// TwinCAT 3 PLC project nadaCAT
// ProgramVersion: 3.1.4024.0
// libraries:
//   Tc2_MC2, * (Beckhoff Automation GmbH)
//   Tc2_MC2_Drive, * (Beckhoff Automation GmbH)
//   Tc2_Standard, * (Beckhoff Automation GmbH)
//   Tc2_System, * (Beckhoff Automation GmbH)
//   Tc2_TcpIp, * (Beckhoff Automation GmbH)
//   Tc2_Utilities, * (Beckhoff Automation GmbH)
//   Tc3_Module, * (Beckhoff Automation GmbH)
//   VisuDialogs, * (System)
//   VisuSymbols,3.5.10.0,System
// project tree:
//   DUTs/Enums/ E_CommandList.TcTLEO, E_ServoState.TcTLEO (not stored), E_TCPState.TcTLEO
//   DUTs/Hardware/ EL1008.TcDUT (not stored), EL2008.TcDUT (not stored)
//   DUTs/Structs/ dutCommand.TcDUT (not stored), dutResponse.TcDUT, mcInterface.TcDUT, mcOutputs.TcDUT, stConfigParams.TcDUT, stIOinput.TcDUT, stIOoutput.TcDUT, stServoInterface.TcDUT, stStateTransitions.TcDUT (not stored)
//   / GlobalTextList.TcGTLO, PlcTask.TcTTO, Visualization Manager.TcVMO (not stored), VISU_TASK.TcTTO (not stored)
//   GVLs/ gvlMotion.TcGVL, gvlIO.TcGVL, gvlSystem.TcGVL, gvlServo.TcGVL (not stored)
//   POUs/FBs/ FB_AutoMotionControl.TcPOU, FB_ManualMotionControl.TcPOU, FB_ManualMotionControlNew.TcPOU, FB_ManualStateMachine.TcPOU (not stored), FB_TCPServer.TcPOU (not stored), sfc_TCPServer.TcPOU (not stored)
//   POUs/ MAIN.TcPOU
//   POUs/PRGs/ prgMotion.TcPOU (not stored), prgIO.TcPOU, prgSystem.TcPOU, prgTCPComm.TcPOU (not stored)
//   VISUs/ Main.TcVIS (not stored)
//   VISUs/Templates/ MotorFaceplate.TcVIS, MotorFaceplate2.TcVIS (not stored), SysPanel.TcVIS (not stored)
// real-time tasks:
//   TASK PlcTask: cycle T#10ms, priority 20, ADS port 350
//   TASK VISU_TASK: cycle T#200000us, priority 30, ADS port 351
// motion (NC):
//   TASK NC-Task 1 SAF: cycle T#2ms, priority 4, ADS port 501
//   TASK NC-Task 1 SVB: cycle T#10ms, priority 8, ADS port 511
//   AXIS Bank1 (id 4)
//     Dynamic: AccelerationMaximum=1000, DecelerationMaximum=1000, Acceleration=250, Deceleration=250, Jerk=1000, FastAcceleration=10000, FastDeceleration=10000, FastJerk=10000
//     Velo: Maximum=450
//     OtherSettings: AllowMotionCmdToSlave=true
//     encoder EncType=19
//       EncPara: ScaleFactorNumerator=10, ScaleFactorDenominator=3600000, Offset=2.25188333333333, Inverse=true, MaxCount=#xffffffff, ReferenceSystem=3
//         SoftEndMinControl: Enable=true
//         SoftEndMaxControl: Enable=true, Range=860
//     drive DrvType=16
//       DrvPara: Inverse=true, MaxCount=#xffffffff, DriveControlDWord=#x00020000
//         Analog: TorqueSetpointScale=10, ScaleFactorActTorque=0.1
//         TimeComp: TaskDelayCycles=1
//     controller CtrType=1
//       CtrPara: PriorControlFactor=1
//         Observer: BandWidth=20
//   AXIS Virtual (id 2)
//     OtherSettings: AllowMotionCmdToSlave=true
//     encoder EncType=1
//       SoftEndMinControl: Enable=true, Range=-0.1
//       SoftEndMaxControl: Enable=true, Range=860
//     drive DrvType=5
//       Analog: TorqueSetpointScale=10, ScaleFactorActTorque=0.1
//       TimeComp: TaskDelayCycles=1
//     controller CtrType=1
//       CtrPara: PriorControlFactor=1
//         Observer: BandWidth=20
// I/O:
//   DEVICE Device 1 (EtherCAT) (disabled), AmsNetId 192.168.5.101.2.1
//     Drive 1 (IndraDrive MPB20/21 CoE) [IndraDrive MPB20/21 CoE]
//       modules: Module 1 (Cyclic sync position mode)
// variable links:
//   NC-Task 1 SAF/Axes/Bank1 <-> Device 1 (EtherCAT)/Drive 1 (IndraDrive MPB20/21 CoE)
//     Drive/Inputs/In/nDcOutputTime <-> InfoData/DcOutputShift
//     Drive/Inputs/In/nState1 <-> Module 1 (Cyclic sync position mode)/Transmit PDO Mapping Parameter/CiA402: Statusword
//     Drive/Inputs/In/nState2 <-> Module 1 (Cyclic sync position mode)/Transmit PDO Mapping Parameter/CiA402: Statusword @bit 8
//     Drive/Inputs/In/nState4 @bit 1 <-> WcState/InputToggle
//     Drive/Inputs/In/nState4 <-> WcState/WcState
//     Drive/Outputs/Out/nCtrl1 <-> Module 1 (Cyclic sync position mode)/Receive PDO Mapping Parameter/CiA402: Controlword
//     Drive/Outputs/Out/nCtrl2 <-> Module 1 (Cyclic sync position mode)/Receive PDO Mapping Parameter/CiA402: Controlword @bit 8
//     Drive/Outputs/Out/nDataOut1 <-> Module 1 (Cyclic sync position mode)/Receive PDO Mapping Parameter/CiA402: Target position
//     Enc/Inputs/In/nDataIn1 <-> Module 1 (Cyclic sync position mode)/Transmit PDO Mapping Parameter/CiA402: Position actual value
//     Enc/Inputs/In/nDcInputTime <-> InfoData/DcInputShift
//     Enc/Inputs/In/nState4 @bit 1 <-> WcState/InputToggle
//     Enc/Inputs/In/nState4 <-> WcState/WcState
//   nadaCAT/nadaCAT Instance <-> NC-Task 1 SAF/Axes/Virtual
//     PlcTask Inputs/ServoGVLs.servo1Interface.ioAxisRef.NcToPlc <-> Outputs/ToPlc
//     PlcTask Outputs/ServoGVLs.servo1Interface.ioAxisRef.PlcToNc <-> Inputs/FromPlc

CONFIGURATION nadaCAT
    RESOURCE PLC ON TwinCAT3
        TASK PlcTask(INTERVAL := T#10ms, PRIORITY := 20);
        PROGRAM MAIN WITH PlcTask : MAIN;
    END_RESOURCE
END_CONFIGURATION

// ---- DUTs/Enums/E_CommandList.TcTLEO
{attribute 'qualified_only'}
{attribute "to_string'}
TYPE E_CommandList :
(
	ERR := -1,
	NULL := 0,
	LIST,
	HOM,
	SCAN,
	MTP,
	MOVA,
	MOVR,
	STAT,
	CALIB,
	PARAM
);
END_TYPE
//  ERR = '-1'

// ---- DUTs/Enums/E_TCPState.TcTLEO
{attribute 'qualified_only'}
{attribute 'strict'}
TYPE E_TCPState :
(
	enum_member := 0
);
END_TYPE

// ---- DUTs/Structs/dutResponse.TcDUT
TYPE dutResponse :
STRUCT
END_STRUCT
END_TYPE

// ---- DUTs/Structs/mcInterface.TcDUT
TYPE mcInterface :
STRUCT
	bBusy				: BOOL;
	bActive				: BOOL;
	bCommandAborted		: BOOL;
	bError				: BOOL;
	iErrorID			: UDINT;
END_STRUCT
END_TYPE

// ---- DUTs/Structs/mcOutputs.TcDUT
TYPE mcOutputs :
STRUCT
	Status			: BOOL;
	Done			: BOOL;
	Busy			: BOOL;
	Active			: BOOL;
	CommandAborted	: BOOL;
	Error			: BOOL;
	ErrorID			: UDINT;
	
END_STRUCT
END_TYPE

// ---- DUTs/Structs/stConfigParams.TcDUT
TYPE stConfigParams :
STRUCT
	iSpeed		: INT;  		// Stocker speed
	iAccel		: INT;  		// Stocker acceleration
	iDecel		: INT;  		// Stocker deceleration
	sRamp		: STRING(255);  // Stocker ramp style
	iPodPos		: INT;  		// Stocker pod position, given pod
	iScStart	: INT;  		// Stocker start scanning position
	iScEnd		: INT;  		// Stocker end scanning position
	iScThick	: INT;  		// Average wafer thickness
	iScExclLo	: INT;  		// Low wafer exclusion zone (in percent)
	iScExclHi	: INT;			// High wafer exclusion zone (in percent)
	iPdSlot		: INT;  		// Pod slot count
	iPdBtm		: INT;  		// Pod bottom slot position
	iPdTop		: INT;  		// Pod top slot position

END_STRUCT
END_TYPE

// ---- DUTs/Structs/stIOinput.TcDUT
TYPE stIOinput :
STRUCT
// ~~~~~ Input Signals ~~~~~
	// Drive CoE
	coeProbe1Signal			: WORD;
	coeProbe1PosLatch		: WORD;
	coeProbe1NegLatch		: WORD;
	
	// Hardware Signals
	Rack1Slot2				: EL1008;
	
END_STRUCT
END_TYPE

// ---- DUTs/Structs/stIOoutput.TcDUT
TYPE stIOoutput :
STRUCT
// ~~~~~ Output Signals ~~~~~
	// Drive CoE
	coeProbingCycleCommand	: WORD;
	coeProbe1Enable			: WORD;
	
	// Hardware Signals
	Rack1Slot2				: EL1008;
END_STRUCT
END_TYPE

// ---- DUTs/Structs/stServoInterface.TcDUT
TYPE stServoInterface :
STRUCT
	/// In_Outs
	ioAxisRef			: Axis_Ref;
	/// Inputs
	bDriveEnable		: BOOL;
	bStopMotion			: BOOL;
	bFaultReset			: BOOL;
	bTriggerMove		: BOOL;
	bJogFWD				: BOOL;
	bJogRev				: BOOL;
	bHome				: BOOL;
	bDemoModeActive		: BOOL;
	bDemoModeStart		: BOOL;
	bDemoModeStop		: BOOL;
	iMotionSelect		: INT;
	rSpeed				: REAL;
	rAccelDecel			: REAL;
	rPosition			: REAL;
	/// Outputs
	bDriveEnabled		: BOOL;
	bStopped			: BOOL;
	bFaulted			: BOOL;
	bMoving				: BOOL;
	bNotMoving			: BOOL;
	bAtHome				: BOOL;
	bAccelerating		: BOOL;
	bDecelerating		: BOOL;
	bDemoModePermissive	: BOOL;
	bInposition			: BOOL;
	bInVelocity			: BOOL;
	rActualSpeed		: REAL;	
	rActualPosition		: REAL;

	
END_STRUCT
END_TYPE

// ---- GVLs/gvlMotion.TcGVL
{attribute 'qualified_only'}
VAR_GLOBAL
// Manual Control
servo1			: FB_ManualMotionControlNew;
bank1			: FB_AutoMotionControl;
manualMode 		: BOOL := TRUE;
autoMode		: BOOL;

// Server Control
cmdData 		: dutCommand;
bEnableDrive	: BOOL := FALSE;
bStartDrive		: BOOL := FALSE;
bTriggerDefault : BOOL := FALSE;
bInterlockOK	: BOOL := TRUE;
mcBankAxis		: stServoInterface;
driveStatus 	: ST_AxisStatus;	
END_VAR

// ---- GVLs/gvlIO.TcGVL
{attribute 'qualified_only'}
VAR_GLOBAL
	/// Inputs
	stInputs	:	stIOinput;
	/// Outputs
	stOutputs	: 	stIOoutput;
	
	bHomeSwitch: BOOL;
END_VAR

// ---- GVLs/gvlSystem.TcGVL
{attribute 'qualified_only'}
VAR_GLOBAL
	iTaskIdx 	: DINT;
	bFirstCycle : BOOL;
END_VAR

// ---- POUs/MAIN.TcPOU
PROGRAM MAIN
VAR

END_VAR

// System Control
gvlSystem.iTaskIdx  := GETCURTASKINDEXEX();
prgSystem(iTaskIdx 	:= gvlSystem.iTaskIdx,
	   bFirstCycle  := gvlSystem.bFirstCycle);

// IO (comment for simulation)
//prgIO();
	   
// TCP Connection
prgTCPComm(cmdData => gvlMotion.cmdData);

// Motion Control
prgMotion(
	cmdData:= gvlMotion.cmdData, 
	bAutoEnableDrive:= gvlMotion.bEnableDrive, 
	bAutoStartDrive:= gvlMotion.bStartDrive, 
	bAutoInterlockOK:= gvlMotion.bInterlockOK, 
	bAutoTriggerDefault:= gvlMotion.bTriggerDefault, 
	autoDriveStatus=> gvlMotion.driveStatus, 
	cmdResponse=>, 
	arrServoInterface:= gvlServo.arrServoInterface);

END_PROGRAM

// ---- POUs/PRGs/prgSystem.TcPOU
PROGRAM prgSystem
VAR_IN_OUT
	iTaskIdx		: DINT;
	bFirstCycle		: BOOL;
END_VAR

// Scan Control
bFirstCycle := TwinCAT_SystemInfoVarList._TaskInfo[iTaskIdx].FirstCycle;

// Mode Control
gvlMotion.autoMode := NOT gvlMotion.manualMode;

END_PROGRAM

// ---- POUs/FBs/FB_ManualMotionControlNew.TcPOU
FUNCTION_BLOCK FB_ManualMotionControlNew
VAR_INPUT
	iCmdMova		:	INT := 0;
	iCmdMovr		: 	INT := 0;
	bEnableDrive	:   BOOL;
	bStartDrive		: 	BOOL;
	bRunOnce		:   BOOL := TRUE;
END_VAR
VAR_OUTPUT
	driveStatus	: ST_AxisStatus;
END_VAR
VAR_IN_OUT
	mcBankAxis	: stServoInterface;
END_VAR

VAR
	eState					: E_ServoState;
	demoState				: FB_ManualStateMachine;
	servoPower				: MC_Power;
	servoBuffer				: MC_BufferMode := MC_Aborting;
	servoReset				: MC_Reset;
	servoHome				: MC_Home;
	servoStatus				: MC_ReadStatus;
	servoSetPosition		: MC_SetPosition;
	servoJog				: MC_Jog;
	servoStop				: MC_Stop;
	servoMoveAbsolute		: MC_MoveAbsolute;
	servoMoveRelative		: MC_MoveRelative;
	servoMoveVelocity		: MC_MoveVelocity;
	jogErrorID				: UDINT;
	errorStop: BOOL;
	disabled: BOOL;
	stopping: BOOL;
	discreteMotion: BOOL;
	continuousMotion: BOOL;
	syncMotion: BOOL;
	homing: BOOL;
	constVelocity: BOOL;
	accel: BOOL;
	decel: BOOL;
	status: ST_AxisStatus;
	powerInterface 		: mcInterface;
	resetInterface		: mcInterface;
	homeInterface		: mcInterface;
	jogInterface		: mcInterface;
	stopInterface		: mcInterface;
	moveAbsInterface	: mcInterface;
	moveRelInterface	: mcInterface;
	moveVelInterface	: mcInterface;
	statusInterface		: mcInterface;
	
	// State Machine Variables
	startCycle			: BOOL;
	continueToTop		: BOOL;
	continueToBottom	: BOOL;
	endAtTop			: BOOL;
	endAtBottom			: BOOL;
	moveBottomTrig			: BOOL;
	moveTopTrig				: BOOL;
	
	demoModePermissive	: BOOL;
	demoModeRun			: BOOL;
	bottomComplete		: BOOL;
	topComplete			: BOOL;
	
	servoMoveBottom		: MC_MoveAbsolute;
	servoMoveTop		: MC_MoveAbsolute;
	servoEstop			: MC_Halt;
	
	demoModePermissivesdf: INT;
END_VAR

// ~~~~ Manual FB Inits ~~~~
// Status
servoStatus(
	Axis:= mcBankAxis.ioAxisRef, 
	Enable:= TRUE, 
	Valid=> , 
	Busy=> statusInterface.bBusy, 
	Error=> statusInterface.bError, 
	ErrorID=> statusInterface.iErrorID, 
	ErrorStop=> errorStop, 
	Disabled=> disabled, 
	Stopping=> stopping, 
	StandStill=> mcBankAxis.bNotMoving, 
	DiscreteMotion=> discreteMotion, 
	ContinuousMotion=> continuousMotion, 
	SynchronizedMotion=> syncMotion, 
	Homing=> homing, 
	ConstantVelocity=> mcBankAxis.bInVelocity, 
	Accelerating=> mcBankAxis.bAccelerating, 
	Decelerating=> mcBankAxis.bDecelerating, 
	Status=> status);

// Enable
servoPower(
	Axis:= mcBankAxis.ioAxisRef, 
	Enable:= mcBankAxis.bDriveEnable, 
	Enable_Positive:=TRUE , 
	Enable_Negative:=TRUE , 
	Override:=100.0 , 
	BufferMode:=servoBuffer , 
	Options:= servoPower.Options, 
	Busy=> powerInterface.bBusy, 
	Active=> powerInterface.bActive, 
	Error=> powerInterface.bError, 
	ErrorID=> powerInterface.iErrorID);
// Init Stop
servoStop(
	Axis:= mcBankAxis.ioAxisRef, 
	Execute:=mcBankAxis.bStopMotion , 
	Deceleration:= 100, 
	Jerk:=100 , 
	Options:= servoStop.Options, 
	Busy=>stopInterface.bBusy , 
	Active=>stopInterface.bActive , 
	CommandAborted=>stopInterface.bCommandAborted , 
	Error=> stopInterface.bError, 
	ErrorID=> stopInterface.iErrorID);

// Init HOM
servoHome(
	Axis:= mcBankAxis.ioAxisRef, 
	Execute:= mcBankAxis.bHome, 
	Position:=0.0 , 
	HomingMode:= MC_DefaultHoming, 
	BufferMode:= servoBuffer, 
	bCalibrationCam:=gvlIO.bHomeSwitch , 
	Busy=>homeInterface.bBusy , 
	Active=> homeInterface.bActive, 
	CommandAborted=>homeInterface.bCommandAborted , 
	Error=>homeInterface.bError , 
	ErrorID=> homeInterface.iErrorID);

// Init JOG
servoJog(
	Axis:= mcBankAxis.ioAxisRef, 
	JogForward:= mcBankAxis.bJogFWD, 
	JogBackwards:= mcBankAxis.bJogRev, 
	Mode:= servoJog.Mode, 
	Position:=5 , 
	Velocity:= 1, 
	Acceleration:= 250, 
	Deceleration:= 250, 
	Jerk:= 5000, 
	Busy=>jogInterface.bBusy , 
	Active=>jogInterface.bActive , 
	CommandAborted=>jogInterface.bCommandAborted , 
	Error=>jogInterface.bError , 
	ErrorID=>jogInterface.iErrorID );


// Init MOVA
servoMoveAbsolute(
	Axis:= mcBankAxis.ioAxisRef, 
	Execute:= (mcBankAxis.bTriggerMove AND (mcBankAxis.iMotionSelect = 1)), 
	Position:= mcBankAxis.rPosition, 
	Velocity:=mcBankAxis.rSpeed , 
	Acceleration:=mcBankAxis.rAccelDecel , 
	Deceleration:= mcBankAxis.rAccelDecel, 
	Jerk:= 500, 
	BufferMode:= servoBuffer, 
	Options:=servoMoveAbsolute.Options , 
	Busy=> moveAbsInterface.bBusy, 
	Active=> moveAbsInterface.bActive, 
	CommandAborted=>moveAbsInterface.bCommandAborted , 
	Error=> moveAbsInterface.bError, 
	ErrorID=> moveAbsInterface.iErrorID);

// Init MovVel
servoMoveVelocity(
	Axis:= mcBankAxis.ioAxisRef, 
	Execute:= (mcBankAxis.bTriggerMove AND (mcBankAxis.iMotionSelect = 3)), 
	Velocity:= mcBankAxis.rSpeed, 
	Acceleration:= mcBankAxis.rAccelDecel, 
	Deceleration:= mcBankAxis.rAccelDecel, 
	Jerk:= 500, 
	Direction:= servoMoveVelocity.Direction, 
	BufferMode:= servoBuffer, 
	Options:= servoMoveVelocity.Options,  
	Busy=> moveVelInterface.bBusy, 
	Active=> moveVelInterface.bActive, 
	CommandAborted=> moveVelInterface.bCommandAborted, 
	Error=>moveVelInterface.bError , 
	ErrorID=> moveVelInterface.iErrorID);
	
// Init Servo Move Top
servoMoveTop(
	Axis:= mcBankAxis.ioAxisRef, 
	Execute:= demoModeRun, 
	Position:= 800, 
	Velocity:= 150, 
	Acceleration:= 1000, 
	Deceleration:= 1000, 
	Jerk:= 1000, 
	BufferMode:= servoBuffer, 
	Options:= servoMoveAbsolute.Options, 
	Done=> topComplete, 
	Busy=> moveAbsInterface.bBusy, 
	Active=> moveAbsInterface.bActive, 
	CommandAborted=> moveAbsInterface.bCommandAborted, 
	Error=> moveAbsInterface.bError, 
	ErrorID=> moveAbsInterface.iErrorID);

// Init Servo Move Bottom
	servoMoveBottom(
	Axis:= mcBankAxis.ioAxisRef, 
	Execute:= demoModeRun, 
	Position:= 800, 
	Velocity:= 150, 
	Acceleration:= 1000, 
	Deceleration:= 1000, 
	Jerk:= 1000, 
	BufferMode:= servoBuffer, 
	Options:= servoMoveAbsolute.Options, 
	Done=> bottomComplete,
	Busy=> moveAbsInterface.bBusy, 
	Active=> moveAbsInterface.bActive, 
	CommandAborted=> moveAbsInterface.bCommandAborted, 
	Error=> moveAbsInterface.bError, 
	ErrorID=> moveAbsInterface.iErrorID);

// Sync Axis
syncAxis();	

// ~~~~~ Demo State Machine ~~~~~
// FB Init
demoState(
	startCycle:= startCycle, 
	continueToTop:= continueToTop, 
	continueToBottom:= continueToBottom, 
	endAtTop:= endAtTop, 
	endAtBottom:= endAtBottom, 
	moveBottom=> moveBottomTrig, 
	moveTop=> moveTopTrig);
	
// Cycle Start
IF demoModePermissive AND demoModeRun THEN
	startCycle := TRUE;
ELSE 
	startCycle := FALSE;
END_IF

// Continue to Top
IF bottomComplete AND demoModeRun THEN
	continueToTop := TRUE;
ELSE
	continueToTop := FALSE;
END_IF


// Continue to Bottom
IF topComplete AND demoModeRun THEN
	continueToBottom := TRUE;
ELSE
	continueToBottom := FALSE;
END_IF

// End at Bottom
IF bottomComplete AND NOT demoModeRun THEN
	endAtBottom := TRUE;
ELSE
	endAtBottom := FALSE;
END_IF

// End at Top
IF topComplete AND demoModeRun THEN
	endAtTop := TRUE;
ELSE
	endAtTop := FALSE;
END_IF

ACTION moveBottom:
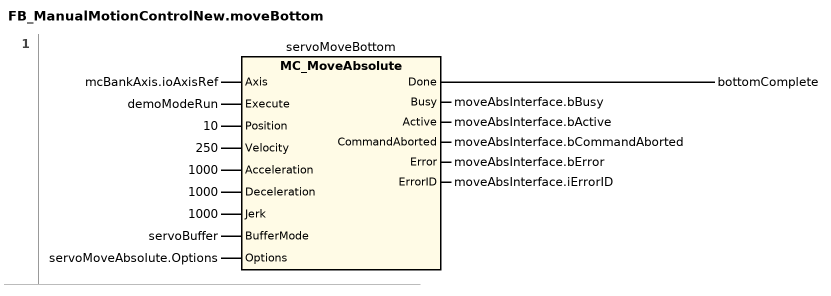
// NETWORK 1
servoMoveBottom(
    Axis := mcBankAxis.ioAxisRef,
    Execute := demoModeRun,
    Position := 10,
    Velocity := 250,
    Acceleration := 1000,
    Deceleration := 1000,
    Jerk := 1000,
    BufferMode := servoBuffer,
    Options := servoMoveAbsolute.Options,
    Busy => moveAbsInterface.bBusy,
    Active => moveAbsInterface.bActive,
    CommandAborted => moveAbsInterface.bCommandAborted,
    Error => moveAbsInterface.bError,
    ErrorID => moveAbsInterface.iErrorID); // MC_MoveAbsolute
bottomComplete := servoMoveBottom.Done;
END_ACTION

ACTION moveTop:
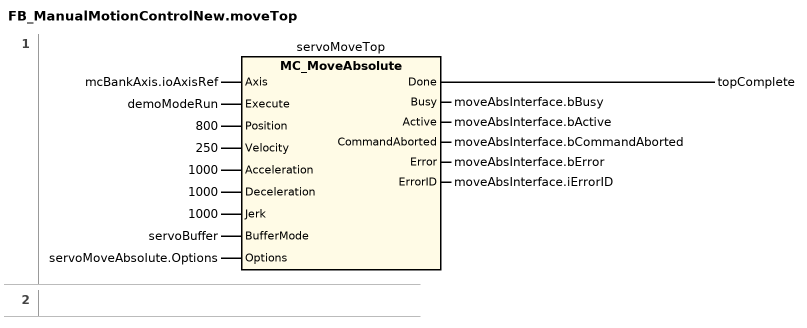
// NETWORK 1
servoMoveTop(
    Axis := mcBankAxis.ioAxisRef,
    Execute := demoModeRun,
    Position := 800,
    Velocity := 250,
    Acceleration := 1000,
    Deceleration := 1000,
    Jerk := 1000,
    BufferMode := servoBuffer,
    Options := servoMoveAbsolute.Options,
    Busy => moveAbsInterface.bBusy,
    Active => moveAbsInterface.bActive,
    CommandAborted => moveAbsInterface.bCommandAborted,
    Error => moveAbsInterface.bError,
    ErrorID => moveAbsInterface.iErrorID); // MC_MoveAbsolute
topComplete := servoMoveTop.Done;

// NETWORK 2
END_ACTION

ACTION syncAxis:
CASE mcBankAxis.ioAxisRef.NcToPlc.AxisState OF
	0 : // Inactive
	
	1 : // Running
		
	3 : // Phase_VeloConst
		mcBankAxis.bInVelocity := TRUE;
	4 : // Phase_AccPos
		mcBankAxis.bAccelerating := TRUE;
	5 : // Phase_AccNeg
		mcBankAxis.bDecelerating := TRUE;
END_CASE

// Feedback

mcBankAxis.rActualPosition := mcBankAxis.ioAxisRef.NcToPlc.ActPos;

mcBankAxis.rActualSpeed := mcBankAxis.ioAxisRef.NcToPlc.ActVelo;

// Motion Status
mcBankAxis.bDriveEnabled:= NOT(disabled);
mcBankAxis.bMoving := NOT(mcBankAxis.bNotMoving AND disabled);
mcBankAxis.bFaulted := statusInterface.bError;

// Drive Control

// Demo Mode
IF mcBankAxis.iMotionSelect = 1 THEN
	demoModePermissive := TRUE;
ELSE
	demoModePermissive := FALSE;
END_IF

IF demoModePermissive AND (mcBankAxis.bDemoModeStart OR demoModeRun) AND NOT mcBankAxis.bDemoModeStop THEN
	demoModeRun := TRUE;
ELSE
	demoModeRun := FALSE;
END_IF
END_ACTION

END_FUNCTION_BLOCK

// ---- POUs/FBs/FB_AutoMotionControl.TcPOU
FUNCTION_BLOCK FB_AutoMotionControl
VAR_INPUT
	cmdData			: 	dutCommand;
	bEnableDrive	:   BOOL;
	bStartDrive		: 	BOOL;
	bInterlockOK	:	BOOL := TRUE;
	bTriggerDefault	: 	BOOL := TRUE;
END_VAR
VAR_OUTPUT
	driveStatus		: ST_AxisStatus;
END_VAR
VAR_IN_OUT
	mcBankAxis		:	stServoInterface;
END_VAR
VAR
	eCommand		: 	E_CommandList;
	rCmdMova		:	REAL := 0.0;
	rCmdMovr		: 	REAL := 0.0;
	bInitialized	: 	BOOL := FALSE;
	eState			: 	E_ServoState := E_ServoState.DEFAULT;
	// Admin Controls
	fbBankStatus	: MC_ReadStatus;
	fbBankEnable	: MC_Power;
	fbBankReset		: MC_Reset;
	mcBufferMode	: MC_BufferMode := MC_BufferMode.MC_Aborting;
	mcOptions 		: ST_PowerOptions;
	powerOutputs	: mcOutputs;
	resetOutputs	: mcOutputs;
	bReset			: BOOL;
	// Homing Controls
	fbBankHome		: MC_Home;
	homeOptions		: ST_HomingOptions;
	dummyCam		: BOOL;
	homeOutputs		: mcOutputs;
	
	// Motion Controls
	dummyRobotClear	: BOOL;
	fbBankMovA		: MC_MoveAbsolute;
	movaOption		: ST_MoveOptions;
	fbBankMovR		: MC_MoveRelative;
	movrOptions		: ST_MoveOptions;
	fbBankStop		: MC_Stop;		
	fbBankHalt		: MC_Halt;
	movaOutputs		: mcOutputs;
	movrOutputs		: mcOutputs;
	stopOutputs		: mcOutputs;
	haltOutputs		: mcOutputs;
	runOnce			: BOOL;	//Oneshot for motion inits
END_VAR

StateMachine();
ServoInit();
IF eState >= E_ServoState.HOMING THEN
	ServoMotion();
END_IF

// Motion Inits

// Status
fbBankStatus(
	Axis:= mcBankAxis.ioAxisRef, 
	Enable:= TRUE, 
	Valid=> , 
	Busy=> , 
	Error=> , 
	ErrorID=> , 
	ErrorStop=> , 
	Disabled=> , 
	Stopping=> , 
	StandStill=> , 
	DiscreteMotion=> , 
	ContinuousMotion=> , 
	SynchronizedMotion=> , 
	Homing=> , 
	ConstantVelocity=> , 
	Accelerating=> , 
	Decelerating=> , 
	Status=> driveStatus);

// Enable
fbBankEnable(AXIS := mcBankAxis.ioAxisRef,
			 Enable_Positive := TRUE,
			 Enable_Negative := TRUE,
			 Override := 100,
			 BufferMode := mcBufferMode,
			 Options := mcOptions,
			 Status => powerOutputs.Status,
			 Busy => powerOutputs.Busy,
			 Active => powerOutputs.Active,
			 Error => powerOutputs.Error,
			 ErrorID => powerOutputs.ErrorID);
// Reset
fbBankReset(Axis:=mcBankAxis.ioAxisRef);
// Stop
fbBankStop(
	Axis:= mcBankAxis.ioAxisRef, 
	Done=> stopOutputs.Done, 
	Busy=> stopOutputs.Busy, 
	Active=> stopOutputs.Active, 
	CommandAborted=> stopOutputs.CommandAborted, 
	Error=> stopOutputs.Error, 
	ErrorID=> stopOutputs.ErrorID);

// Init HOM
fbBankHome(
	Axis:= mcBankAxis.ioAxisRef, 
	Position:= DEFAULT_HOME_POSITION, 
	HomingMode:= MC_DefaultHoming, 
	BufferMode:= mcBufferMode, 
	Options:= homeOptions, 
	bCalibrationCam:= (ABS(mcBankAxis.rActualPosition) <= 0.001), 
	Done=> homeOutputs.Done, 
	Busy=> homeOutputs.Busy, 
	Active=> homeOutputs.Active, 
	CommandAborted=> homeOutputs.CommandAborted, 
	Error=> homeOutputs.Error, 
	ErrorID=> homeOutputs.ErrorID);

// Init MOVA
fbBankMovA(
	Axis:= mcBankAxis.ioAxisRef, 
	Position:= rCmdMova, 
	Velocity:= 200, 
	BufferMode:= mcBufferMode, 
	Options:= movaOption, 
	Done=> movaOutputs.Done, 
	Busy=> movaOutputs.Busy, 
	Active=> movaOutputs.Active, 
	CommandAborted=> movaOutputs.CommandAborted, 
	Error=> movaOutputs.Error, 
	ErrorID=> movaOutputs.ErrorID);

// Init MOVR
fbBankMovR(
	Axis:= mcBankAxis.ioAxisRef, 
	Distance:= rCmdMovr, 
	Velocity:= 200, 
	BufferMode:= mcBufferMode, 
	Options:= movrOptions, 
	Done=> movrOutputs.Done, 
	Busy=> movrOutputs.Busy, 
	Active=> movrOutputs.Active, 
	CommandAborted=> movrOutputs.CommandAborted, 
	Error=> movrOutputs.Error, 
	ErrorID=> movrOutputs.ErrorID);

METHOD ServoInit : BOOL
VAR_INPUT
END_VAR
eCommand := cmdData.eCommand;

CASE eState OF
	E_ServoState.DEFAULT:
		
		bTriggerDefault := FALSE;
		bInitialized	:= TRUE;

	E_ServoState.OFF, E_ServoState.DISABLED:
		fbBankEnable.Enable := FALSE;
		fbBankHome.Execute  := FALSE;
		fbBankMovA.Execute  := FALSE;
		fbBankMovR.Execute	:= FALSE;
    
    E_ServoState.ENABLED:
		fbBankEnable.Enable := bStartDrive AND bEnableDrive;
		// Check w/ TCP to ensure buffer is clear
		
	E_ServoState.STANDBY:
		IF eCommand = E_CommandList.MOVA THEN
			rCmdMova := LINT_TO_REAL(cmdData.arrParam[1])/1000.0;
			eState := E_ServoState.MOVE_ABS;
		ELSIF eCommand = E_CommandList.MOVR THEN
			rCmdMovr := LINT_TO_REAL(cmdData.arrParam[1])/1000.0;
			eState := E_ServoState.MOVE_REL;
		ELSIF eCommand = E_CommandList.SCAN THEN
			eState := E_ServoState.MOVE_SCAN;
		END_IF
	
	E_ServoState.FAULTED:
		fbBankReset.Execute := bReset;
    
	E_ServoState.HOMING:
		fbBankHome.Execute := TRUE;
		
		IF homeOutputs.Error THEN
			eState := E_ServoState.FAULTED;
		ELSE
			IF homeOutputs.Active THEN
				IF driveStatus.Homed THEN
					fbBankHome.Execute := FALSE; // Stop homing once complete
					eState := E_ServoState.STANDBY;
				END_IF
			END_IF
		END_IF
END_CASE
END_METHOD

METHOD ServoMotion : BOOL
VAR_INPUT
END_VAR
VAR_IN_OUT
END_VAR
VAR
END_VAR
IF eState <> E_ServoState.INTERLOCK_MOTION THEN
	CASE eState OF

		E_ServoState.HOMING:
			fbBankHome.Execute := NOT (driveStatus.Moving OR driveStatus.Error);

		E_ServoState.MOVE_ABS:
			fbBankMovA.Position := rCmdMova;
			fbBankMovA.Execute := NOT (driveStatus.Moving OR driveStatus.Error);
		
		E_ServoState.MOVE_REL:
			fbBankMovR.Distance := rCmdMovr;
			fbBankMovR.Execute := NOT (driveStatus.Moving OR driveStatus.Error);  // Trigger true until movement detected
			
		E_ServoState.MOVE_SCAN:
			// Handle multiple scan input types
			// SCAN (no parameters), full range
			// SCAN 0, full range
			// SCAN 1, scan position 1
			// SCAN 1,13 scan from position 1 to 13
	END_CASE
ELSIF eState = E_ServoState.INTERLOCK_MOTION THEN
    fbBankStop.Execute := NOT (driveStatus.Moving);
END_IF
END_METHOD

METHOD StateMachine : BOOL
VAR_INPUT
END_VAR
// Interrupt
IF gvlMotion.manualMode THEN
	eState := E_ServoState.OFF;
END_IF

// State Machine
CASE eState OF
    E_ServoState.DEFAULT:
		IF bInitialized THEN
			eState := E_ServoState.DISABLED;
		END_IF
	E_ServoState.OFF:
        IF NOT gvlMotion.manualMode THEN
			eState := E_ServoState.DEFAULT;
		END_IF

    E_ServoState.DISABLED:
		
		IF bEnableDrive AND NOT (driveStatus.Error) THEN
            eState := E_ServoState.ENABLED;
        ELSIF driveStatus.Error THEN
            eState := E_ServoState.FAULTED;
        END_IF
		

    
    E_ServoState.ENABLED:

		IF bStartDrive AND fbBankEnable.Status AND NOT driveStatus.Error THEN
            eState := E_ServoState.STANDBY;
        ELSIF driveStatus.Error THEN
            eState := E_ServoState.FAULTED;
        END_IF
		
        // Placeholder for TCP check

    E_ServoState.STANDBY:
		IF eCommand = E_CommandList.HOM THEN
            eState := E_ServoState.HOMING;
		ELSIF eCommand = E_CommandList.MOVA THEN
			eState := E_ServoState.MOVE_ABS;
		ELSIF eCommand = E_CommandList.MOVR THEN
			eState := E_ServoState.MOVE_REL;
		END_IF
	
	E_ServoState.HOMING:
			IF driveStatus.Error THEN
				eState := E_ServoState.FAULTED;
			ELSIF driveStatus.Homed THEN
				eState := E_ServoState.STANDBY;
			END_IF

	E_ServoState.MOVE_ABS:
		IF driveStatus.InTargetPosition THEN
			eState := E_ServoState.STANDBY;
		END_IF
		IF driveStatus.Error THEN
			eState := E_ServoState.FAULTED;
		END_IF
	
	E_ServoState.MOVE_REL:
		IF driveStatus.InTargetPosition THEN
			eState := E_ServoState.STANDBY;
		END_IF
		IF driveStatus.Error THEN
			eState := E_ServoState.FAULTED;
		END_IF
	
	E_ServoState.INTERLOCK_MOTION:
		IF bInterlockOK AND driveStatus.NotMoving THEN
        	eState := E_ServoState.STANDBY; // Return to standby if motion has stopped
    	END_IF
	E_ServoState.FAULTED:
	
		IF NOT driveStatus.Error THEN
			IF driveStatus.Disabled THEN
				eState := E_ServoState.DISABLED;
			ELSIF driveStatus.Error THEN
				eState := E_ServoState.FAULTED;
			ELSIF driveStatus.Homing THEN
				eState := E_ServoState.HOMING;
			ELSIF driveStatus.NotMoving THEN
				eState := E_ServoState.STANDBY;
			END_IF
		END_IF
		
//        // Catch-all case to prevent transition to DEFAULT unexpectedly
//        eState := E_ServoState.STANDBY;  // Default safe state
//        // Add a debug output here if necessary to track transitions
//        fbBankStatus.Enable := FALSE;  // Explicitly disable status polling if entering an invalid state
END_CASE
END_METHOD

END_FUNCTION_BLOCK

// ---- POUs/FBs/FB_ManualMotionControl.TcPOU
FUNCTION_BLOCK FB_ManualMotionControl
VAR_INPUT
	
END_VAR
VAR_OUTPUT
END_VAR
VAR_IN_OUT
	stServoInterface		: stServoInterface;
END_VAR
VAR
	
	servoPower				: MC_Power;
	servoBuffer				: MC_BufferMode := MC_Aborting;
	
	servoReset				: MC_Reset;
	servoHome				: MC_Home;
	
	servoStatus				: MC_ReadStatus;
	
	servoSetPosition		: MC_SetPosition;
	
	servoJog				: MC_Jog;
	
	servoStop				: MC_Stop;
	
	servoMoveAbsolute		: MC_MoveAbsolute;
	
	servoMoveRelative		: MC_MoveRelative;
	
	servoMoveVelocity		: MC_MoveVelocity;
	
	jogErrorID				: UDINT;
	
	errorStop: BOOL;
	disabled: BOOL;
	stopping: BOOL;
	discreteMotion: BOOL;
	continuousMotion: BOOL;
	syncMotion: BOOL;
	homing: BOOL;
	constVelocity: BOOL;
	accel: BOOL;
	decel: BOOL;
	status: ST_AxisStatus;
	
	powerInterface 		: mcInterface;
	resetInterface		: mcInterface;
	homeInterface		: mcInterface;
	jogInterface		: mcInterface;
	stopInterface		: mcInterface;
	moveAbsInterface	: mcInterface;
	moveRelInterface	: mcInterface;
	moveVelInterface	: mcInterface;
	statusInterface		: mcInterface;
	
	// State Machine Variables
	startCycle			: BOOL;
	continueToTop		: BOOL;
	continueToBottom	: BOOL;
	endAtTop			: BOOL;
	endAtBottom			: BOOL;
	moveBottomTrig			: BOOL;
	moveTopTrig				: BOOL;
	
	demoState			: FB_ManualStateMachine;
	demoModePermissive	: BOOL;
	demoModeRun			: BOOL;
	bottomComplete		: BOOL;
	topComplete			: BOOL;
	
	servoMoveBottom		: MC_MoveAbsolute;
	servoMoveTop		: MC_MoveAbsolute;
	servoEstop			: MC_Halt;
	
	demoModePermissivesdf: INT;
END_VAR

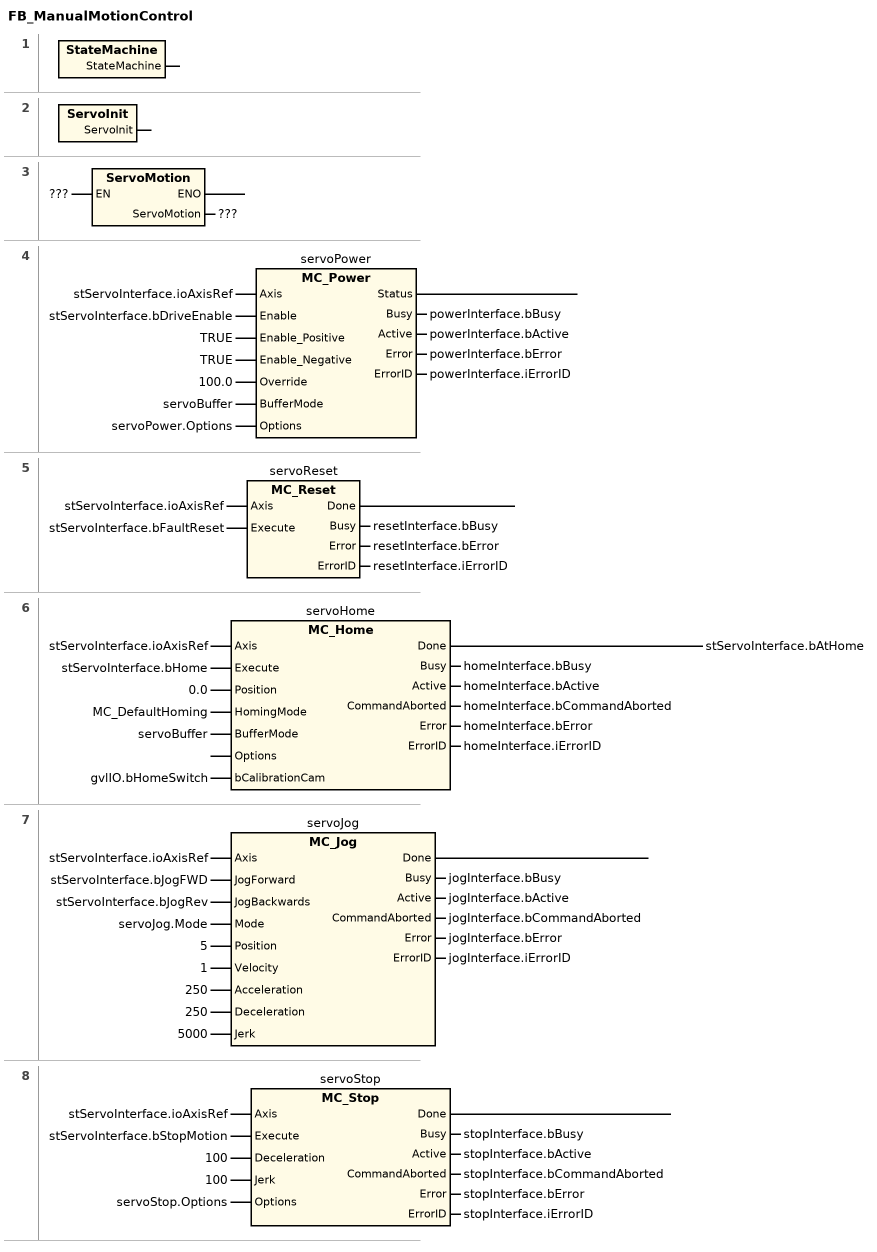
// NETWORK 1
StateMachine();

// NETWORK 2
ServoInit();

// NETWORK 3
ServoMotion();

// NETWORK 4
servoPower(
    Axis := stServoInterface.ioAxisRef,
    Enable := stServoInterface.bDriveEnable,
    Enable_Positive := TRUE,
    Enable_Negative := TRUE,
    Override := 100.0,
    BufferMode := servoBuffer,
    Options := servoPower.Options,
    Busy => powerInterface.bBusy,
    Active => powerInterface.bActive,
    Error => powerInterface.bError,
    ErrorID => powerInterface.iErrorID); // MC_Power

// NETWORK 5
servoReset(
    Axis := stServoInterface.ioAxisRef,
    Execute := stServoInterface.bFaultReset,
    Busy => resetInterface.bBusy,
    Error => resetInterface.bError,
    ErrorID => resetInterface.iErrorID); // MC_Reset

// NETWORK 6
servoHome(
    Axis := stServoInterface.ioAxisRef,
    Execute := stServoInterface.bHome,
    Position := 0.0,
    HomingMode := MC_DefaultHoming,
    BufferMode := servoBuffer,
    bCalibrationCam := gvlIO.bHomeSwitch,
    Busy => homeInterface.bBusy,
    Active => homeInterface.bActive,
    CommandAborted => homeInterface.bCommandAborted,
    Error => homeInterface.bError,
    ErrorID => homeInterface.iErrorID); // MC_Home
stServoInterface.bAtHome := servoHome.Done;

// NETWORK 7
servoJog(
    Axis := stServoInterface.ioAxisRef,
    JogForward := stServoInterface.bJogFWD,
    JogBackwards := stServoInterface.bJogRev,
    Mode := servoJog.Mode,
    Position := 5,
    Velocity := 1,
    Acceleration := 250,
    Deceleration := 250,
    Jerk := 5000,
    Busy => jogInterface.bBusy,
    Active => jogInterface.bActive,
    CommandAborted => jogInterface.bCommandAborted,
    Error => jogInterface.bError,
    ErrorID => jogInterface.iErrorID); // MC_Jog

// NETWORK 8
servoStop(
    Axis := stServoInterface.ioAxisRef,
    Execute := stServoInterface.bStopMotion,
    Deceleration := 100,
    Jerk := 100,
    Options := servoStop.Options,
    Busy => stopInterface.bBusy,
    Active => stopInterface.bActive,
    CommandAborted => stopInterface.bCommandAborted,
    Error => stopInterface.bError,
    ErrorID => stopInterface.iErrorID); // MC_Stop

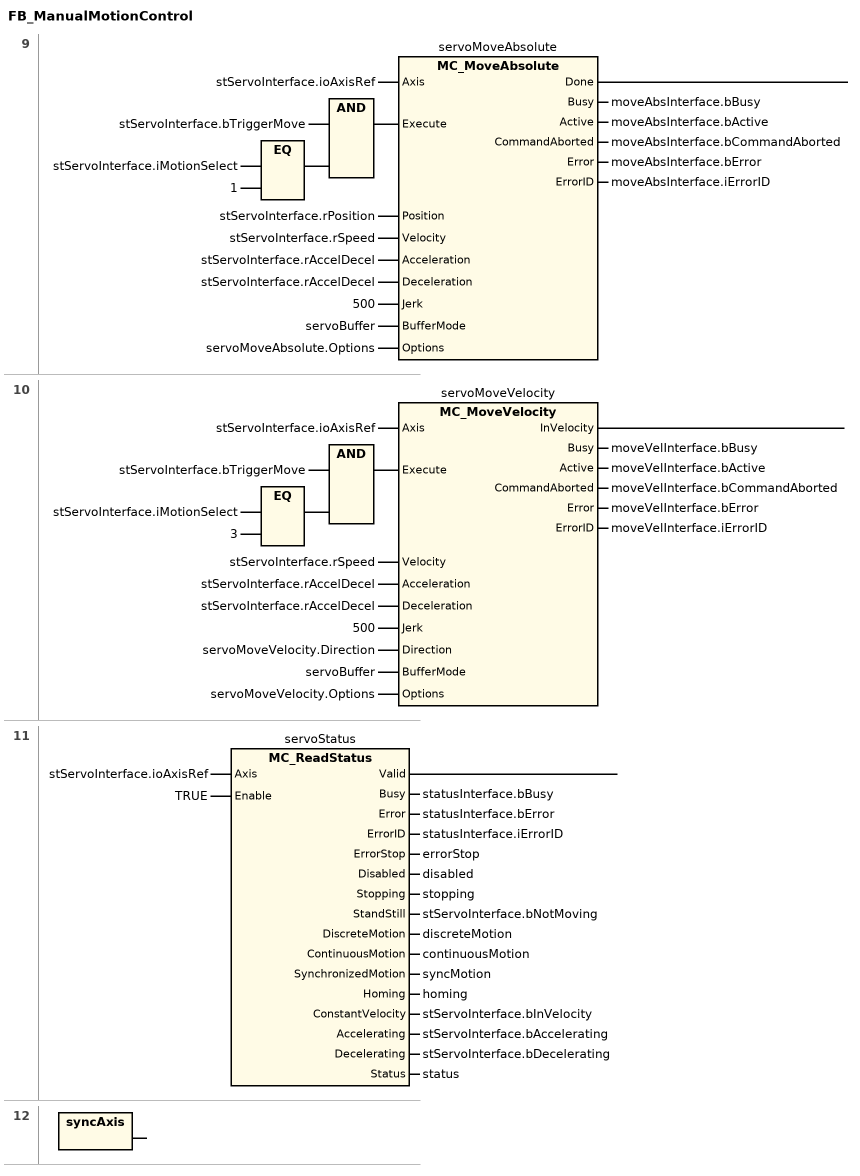
// NETWORK 9
servoMoveAbsolute(
    Axis := stServoInterface.ioAxisRef,
    Execute := stServoInterface.bTriggerMove AND stServoInterface.iMotionSelect = 1,
    Position := stServoInterface.rPosition,
    Velocity := stServoInterface.rSpeed,
    Acceleration := stServoInterface.rAccelDecel,
    Deceleration := stServoInterface.rAccelDecel,
    Jerk := 500,
    BufferMode := servoBuffer,
    Options := servoMoveAbsolute.Options,
    Busy => moveAbsInterface.bBusy,
    Active => moveAbsInterface.bActive,
    CommandAborted => moveAbsInterface.bCommandAborted,
    Error => moveAbsInterface.bError,
    ErrorID => moveAbsInterface.iErrorID); // MC_MoveAbsolute

// NETWORK 10
servoMoveVelocity(
    Axis := stServoInterface.ioAxisRef,
    Execute := stServoInterface.bTriggerMove AND stServoInterface.iMotionSelect = 3,
    Velocity := stServoInterface.rSpeed,
    Acceleration := stServoInterface.rAccelDecel,
    Deceleration := stServoInterface.rAccelDecel,
    Jerk := 500,
    Direction := servoMoveVelocity.Direction,
    BufferMode := servoBuffer,
    Options := servoMoveVelocity.Options,
    Busy => moveVelInterface.bBusy,
    Active => moveVelInterface.bActive,
    CommandAborted => moveVelInterface.bCommandAborted,
    Error => moveVelInterface.bError,
    ErrorID => moveVelInterface.iErrorID); // MC_MoveVelocity

// NETWORK 11
servoStatus(
    Axis := stServoInterface.ioAxisRef,
    Enable := TRUE,
    Busy => statusInterface.bBusy,
    Error => statusInterface.bError,
    ErrorID => statusInterface.iErrorID,
    ErrorStop => errorStop,
    Disabled => disabled,
    Stopping => stopping,
    StandStill => stServoInterface.bNotMoving,
    DiscreteMotion => discreteMotion,
    ContinuousMotion => continuousMotion,
    SynchronizedMotion => syncMotion,
    Homing => homing,
    ConstantVelocity => stServoInterface.bInVelocity,
    Accelerating => stServoInterface.bAccelerating,
    Decelerating => stServoInterface.bDecelerating,
    Status => status); // MC_ReadStatus

// NETWORK 12
syncAxis();

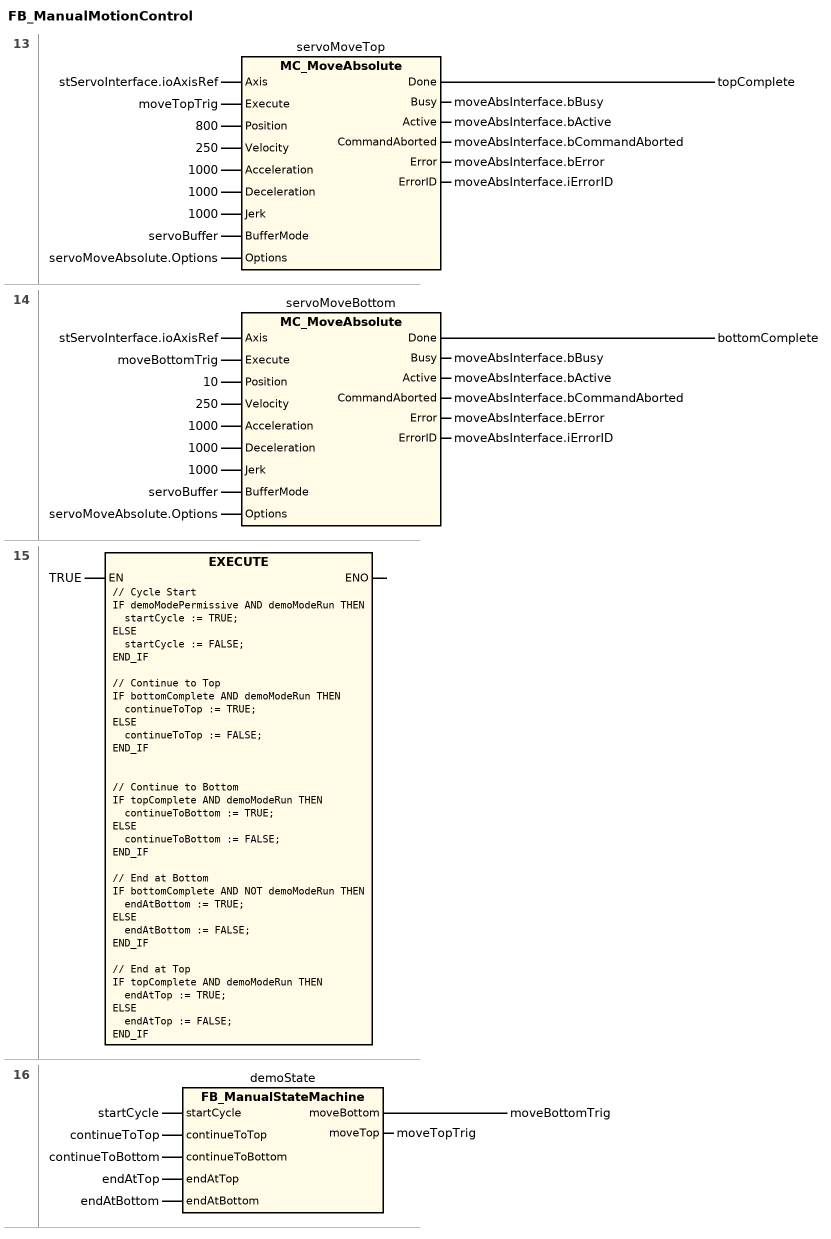
// NETWORK 13
servoMoveTop(
    Axis := stServoInterface.ioAxisRef,
    Execute := moveTopTrig,
    Position := 800,
    Velocity := 250,
    Acceleration := 1000,
    Deceleration := 1000,
    Jerk := 1000,
    BufferMode := servoBuffer,
    Options := servoMoveAbsolute.Options,
    Busy => moveAbsInterface.bBusy,
    Active => moveAbsInterface.bActive,
    CommandAborted => moveAbsInterface.bCommandAborted,
    Error => moveAbsInterface.bError,
    ErrorID => moveAbsInterface.iErrorID); // MC_MoveAbsolute
topComplete := servoMoveTop.Done;

// NETWORK 14
servoMoveBottom(
    Axis := stServoInterface.ioAxisRef,
    Execute := moveBottomTrig,
    Position := 10,
    Velocity := 250,
    Acceleration := 1000,
    Deceleration := 1000,
    Jerk := 1000,
    BufferMode := servoBuffer,
    Options := servoMoveAbsolute.Options,
    Busy => moveAbsInterface.bBusy,
    Active => moveAbsInterface.bActive,
    CommandAborted => moveAbsInterface.bCommandAborted,
    Error => moveAbsInterface.bError,
    ErrorID => moveAbsInterface.iErrorID); // MC_MoveAbsolute
bottomComplete := servoMoveBottom.Done;

// NETWORK 15
// Cycle Start
IF demoModePermissive AND demoModeRun THEN
	startCycle := TRUE;
ELSE 
	startCycle := FALSE;
END_IF

// Continue to Top
IF bottomComplete AND demoModeRun THEN
	continueToTop := TRUE;
ELSE
	continueToTop := FALSE;
END_IF


// Continue to Bottom
IF topComplete AND demoModeRun THEN
	continueToBottom := TRUE;
ELSE
	continueToBottom := FALSE;
END_IF

// End at Bottom
IF bottomComplete AND NOT demoModeRun THEN
	endAtBottom := TRUE;
ELSE
	endAtBottom := FALSE;
END_IF

// End at Top
IF topComplete AND demoModeRun THEN
	endAtTop := TRUE;
ELSE
	endAtTop := FALSE;
END_IF

// NETWORK 16
demoState(
    startCycle := startCycle,
    continueToTop := continueToTop,
    continueToBottom := continueToBottom,
    endAtTop := endAtTop,
    endAtBottom := endAtBottom,
    moveTop => moveTopTrig); // FB_ManualStateMachine
moveBottomTrig := demoState.moveBottom;

ACTION moveBottom:
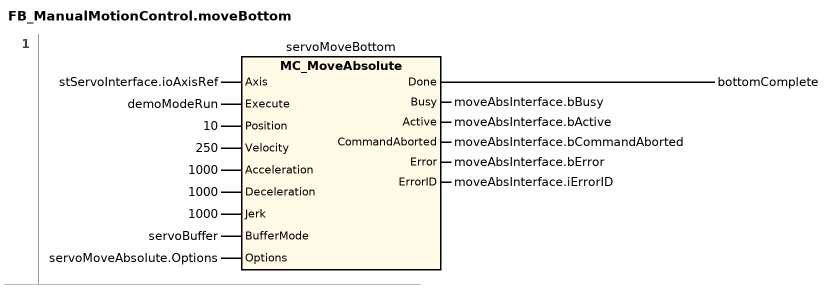
// NETWORK 1
servoMoveBottom(
    Axis := stServoInterface.ioAxisRef,
    Execute := demoModeRun,
    Position := 10,
    Velocity := 250,
    Acceleration := 1000,
    Deceleration := 1000,
    Jerk := 1000,
    BufferMode := servoBuffer,
    Options := servoMoveAbsolute.Options,
    Busy => moveAbsInterface.bBusy,
    Active => moveAbsInterface.bActive,
    CommandAborted => moveAbsInterface.bCommandAborted,
    Error => moveAbsInterface.bError,
    ErrorID => moveAbsInterface.iErrorID); // MC_MoveAbsolute
bottomComplete := servoMoveBottom.Done;
END_ACTION

ACTION moveTop:
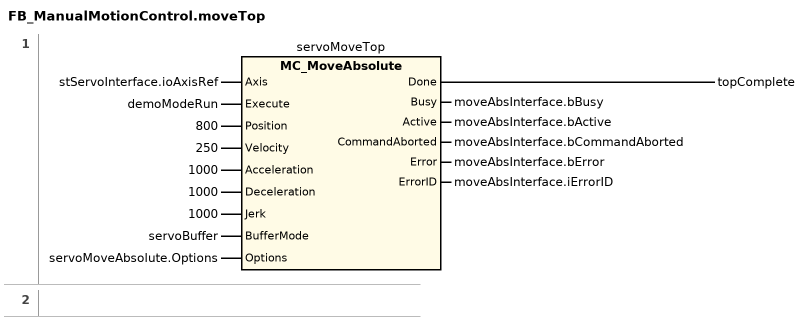
// NETWORK 1
servoMoveTop(
    Axis := stServoInterface.ioAxisRef,
    Execute := demoModeRun,
    Position := 800,
    Velocity := 250,
    Acceleration := 1000,
    Deceleration := 1000,
    Jerk := 1000,
    BufferMode := servoBuffer,
    Options := servoMoveAbsolute.Options,
    Busy => moveAbsInterface.bBusy,
    Active => moveAbsInterface.bActive,
    CommandAborted => moveAbsInterface.bCommandAborted,
    Error => moveAbsInterface.bError,
    ErrorID => moveAbsInterface.iErrorID); // MC_MoveAbsolute
topComplete := servoMoveTop.Done;

// NETWORK 2
END_ACTION

METHOD ServoInit : BOOL
VAR_INPUT
END_VAR
END_METHOD

METHOD ServoMotion : BOOL
VAR_INPUT
END_VAR
END_METHOD

METHOD StateMachine : BOOL
VAR_INPUT
END_VAR
END_METHOD

ACTION syncAxis:
CASE stServoInterface.ioAxisRef.NcToPlc.AxisState OF
	0 : // Inactive
	
	1 : // Running
		
	3 : // Phase_VeloConst
		stServoInterface.bInVelocity := TRUE;
	4 : // Phase_AccPos
		stServoInterface.bAccelerating := TRUE;
	5 : // Phase_AccNeg
		stServoInterface.bDecelerating := TRUE;
END_CASE

// Feedback

stServoInterface.rActualPosition := stServoInterface.ioAxisRef.NcToPlc.ActPos;

stServoInterface.rActualSpeed := stServoInterface.ioAxisRef.NcToPlc.ActVelo;

// Motion Status
stServoInterface.bDriveEnabled:= NOT(disabled);
stServoInterface.bMoving := NOT(stServoInterface.bNotMoving AND disabled);
stServoInterface.bFaulted := statusInterface.bError;

// Drive Control

// Demo Mode
IF stServoInterface.iMotionSelect = 1 THEN
	demoModePermissive := TRUE;
ELSE
	demoModePermissive := FALSE;
END_IF

IF demoModePermissive AND (stServoInterface.bDemoModeStart OR demoModeRun) AND NOT stServoInterface.bDemoModeStop THEN
	demoModeRun := TRUE;
ELSE
	demoModeRun := FALSE;
END_IF
END_ACTION

END_FUNCTION_BLOCK

// ---- POUs/PRGs/prgIO.TcPOU
PROGRAM prgIO
VAR;
END_VAR

// ~~~~~ CoE I/O ~~~~~
(*
PLC Inputs

0x2191:01 (bit 0) Probe 1 signal
0x2199:01 Probe 1 positive latched
0x219A:01 Probe 1 negative latched

PLC Outputs

0x20AA:01 Probing cycle command
0x2195:01 Probe 1 enable
*)

// Scan Toggle
gvlServo.bExecute := NOT gvlServo.bExecute;

// ~ Inputs ~
// Probe 1 Signal : 2191:01
gvlServo.coeRead(Axis:= gvlServo.servo1Interface.ioAxisRef,
				  Index := 16#2191,
				  SubIndex := 16#01,
				  Execute := gvlServo.bExecute,
				  Busy =>,
				  pDstBuf := ADR(gvlIO.stInputs.coeProbe1Signal),
				  BufLen := SIZEOF(gvlIO.stInputs.coeProbe1Signal));

// Probe 1 Positive Latched: 2199:01
gvlServo.coeRead(Axis:= gvlServo.servo1Interface.ioAxisRef,
				  Index := 16#2199,
				  SubIndex := 16#01,
				  Execute := gvlServo.bExecute,
				  Busy =>,
				  pDstBuf := ADR(gvlIO.stInputs.coeProbe1PosLatch),
				  BufLen := SIZEOF(gvlIO.stInputs.coeProbe1PosLatch));

// Probe 1 Negative Latched: 219A:01
gvlServo.coeRead(Axis:= gvlServo.servo1Interface.ioAxisRef,
				  Index := 16#219A,
				  SubIndex := 16#01,
				  Execute := gvlServo.bExecute,
				  Busy =>,
				  pDstBuf := ADR(gvlIO.stInputs.coeProbe1NegLatch),
				  BufLen := SIZEOF(gvlIO.stInputs.coeProbe1NegLatch));

// ~ Outputs ~
// Probing Cycle Command : 20AA:01
	gvlServo.coeWrite(
		Axis:= gvlServo.servo1Interface.ioAxisRef, 
		Index:= 16#20AA, 
		SubIndex:= 16#01, 
		pSrcBuf:= ADR(gvlIO.stOutputs.coeProbingCycleCommand), 
		BufLen:= SIZEOF(gvlIO.stOutputs.coeProbingCycleCommand), 
		Execute:= gvlServo.bExecute);
// Probe 1 Enable : 2195:01
	gvlServo.coeWrite(
		Axis:= gvlServo.servo1Interface.ioAxisRef, 
		Index:= 16#2195, 
		SubIndex:= 16#01, 
		pSrcBuf:= ADR(gvlIO.stOutputs.coeProbe1Enable), 
		BufLen:= SIZEOF(gvlIO.stOutputs.coeProbingCycleCommand), 
		Execute:= gvlServo.bExecute);

END_PROGRAM

// ---- GlobalTextList.TcGTLO
TEXTLIST GlobalTextList
  94 = ''
  613 = '!'
  786 = '%.0f'
  760 = 'ABSOLUTE POSITION'
  424 = 'ACCEL/DECEL'
  653 = 'ACCELERATING'
  471 = 'ACTUAL POSITION'
  549 = 'ACTUAL SPEED'
  492 = 'ACUTAL SPEED'
  532 = 'AUTO'
  654 = 'DECELERATING'
  593 = 'Demo Mode'
  490 = 'DEMO MODE'
  268 = 'Demo Start'
  258 = 'Demo Stop'
  116 = 'Drive 1'
  76 = 'Drive 1: Manual Control'
  476 = 'Drive 2'
  434 = 'Drive Control'
  188 = 'DRIVE ENABLE'
  6 = 'Emergency Stop'
  42 = 'FAULT RESET'
  157 = 'Feedback'
  452 = 'GroupBox'
  945 = 'HOME'
  770 = 'IN POSITION'
  667 = 'IN VELOCITY'
  151 = 'JOG'
  902 = 'Jog FWD'
  411 = 'Jog REV'
  683 = 'MANUAL'
  211 = 'Mode Control'
  481 = 'Motion Select'
  856 = 'Motion Status'
  529 = 'MOVING'
  926 = 'NOT MOVING'
  470 = 'POSITION'
  44 = 'RELATIVE POSITION'
  404 = 'Setpoints'
  917 = 'SPEED'
  54 = 'STOP MOTION'
  940 = 'Trigger Move'
  652 = 'VELOCITY CONTROL'
  530 = 'VELOCITY CONTROL;'
END_TEXTLIST

// ---- VISUs/Templates/MotorFaceplate.TcVIS
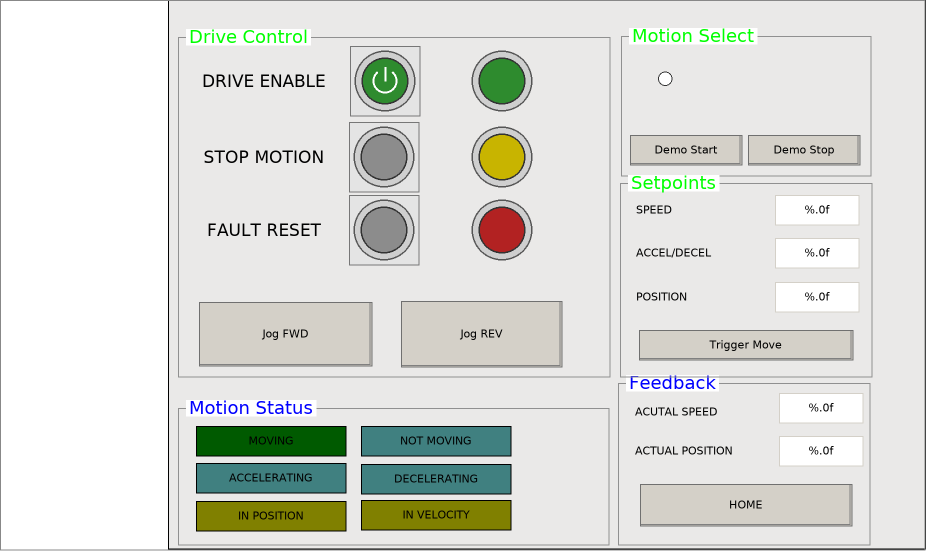
VISUALIZATION MotorFaceplate  // 926x551
    Rectangle (168,-2 758x551)
    GroupBox (178,29 432x348), "Drive Control"
        PowerSwitch (172,17 70x70), variable: gvlServo.servo1Interface.bDriveEnable, behaviour: TOGGLE, style: Switch-PowerSwitch-Green
        PushSwitch (171,93 70x70), variable: gvlServo.servo1Interface.bStopMotion, behaviour: TAP, style: Switch-PushSwitch-Gray
        PushSwitch (171,166 70x70), variable: gvlServo.servo1Interface.bFaultReset, behaviour: TAP, style: Switch-PushSwitch-Gray
        Lamp1 (289,17 70x70), variable: gvlServo.servo1Interface.bDriveEnabled, style: Lamp-Lamp1-Green
        Lamp1 (289,93 70x70), variable: gvlServo.servo1Interface.bNotMoving, style: Lamp-Lamp1-Yellow
        Lamp1 (289,166 70x70), variable: gvlServo.servo1Interface.bFaulted, style: Lamp-Lamp1-Red
        Label (11,37 150x30), "DRIVE ENABLE"
        Label (11,113 150x30), "STOP MOTION"
        Label (11,186 150x30), "FAULT RESET"
        Button (21,273 173x64), "Jog FWD"
            tap gvlServo.servo1Interface.bJogFWD
        Button (223,272 161x66), "Jog REV"
            tap gvlServo.servo1Interface.bJogRev
    GroupBox (178,400 431x145), "Motion Status"
        RoundedRectangle (18,26 150x30), "MOVING", colour toggle: gvlServo.servo1Interface.bMoving
        RoundedRectangle (183,26 150x30), "NOT MOVING", colour toggle: gvlServo.servo1Interface.bNotMoving
        RoundedRectangle (18,63 150x30), "ACCELERATING", colour toggle: gvlServo.servo1Interface.bAccelerating
        RoundedRectangle (183,64 150x30), "DECELERATING", colour toggle: gvlServo.servo1Interface.bDecelerating
        RoundedRectangle (18,101 150x30), "IN POSITION", colour toggle: gvlServo.servo1Interface.bInposition
        RoundedRectangle (183,100 150x30), "IN VELOCITY", colour toggle: gvlServo.servo1Interface.bInVelocity
    GroupBox (618,375 252x170), "Feedback"
        Textfield (161,18 84x30), "%.0f", text variable: gvlServo.servo1Interface.rActualSpeed
        Label (14,61 120x30), "ACTUAL POSITION"
        Textfield (161,61 84x30), "%.0f", text variable: gvlServo.servo1Interface.rActualPosition
        Label (14,22 108x30), "ACUTAL SPEED"
        Button (22,109 212x42), "HOME", invisible if: TRUE
            tap gvlServo.servo1Interface.bHome
    GroupBox (621,28 250x148), "Motion Select"
        RadioButton (35,21 173x59), variable: gvlServo.servo1Interface.iMotionSelect
            p3123465237: DEMO MODE
            p2481256679: RELATIVE POSITION
            p1032612214: VELOCITY CONTROL
        Button (9,107 112x30), "Demo Start", invisible if: gvlServo.servo1Interface.iMotionSelect = 0
            tap gvlServo.servo1Interface.bDemoModeStart
        Button (127,107 112x30), "Demo Stop", invisible if: gvlServo.servo1Interface.iMotionSelect = 0
            tap gvlServo.servo1Interface.bDemoModeStop
    GroupBox (620,175 252x202), "Setpoints"
        Label (13,20 76x30), "SPEED", invisible if: TRUE
        Textfield (155,20 84x30), "%.0f", text variable: gvlServo.servo1Interface.rSpeed, invisible if: TRUE
        Label (13,63 99x30), "ACCEL/DECEL", invisible if: TRUE
        Textfield (155,63 84x30), "%.0f", text variable: gvlServo.servo1Interface.rAccelDecel, invisible if: TRUE
        Label (13,107 76x30), "POSITION", invisible if: TRUE
        Textfield (155,107 84x30), "%.0f", text variable: gvlServo.servo1Interface.rPosition, invisible if: TRUE
        Button (19,155 214x30), "Trigger Move", invisible if: TRUE
            tap gvlServo.servo1Interface.bTriggerMove
END_VISUALIZATION
